% RSLogix 500 project Project6-HourMeter.RSS, saved by version 8.30.00.16 %
PROJECT "UNTITLED"    % processor: Bul.1763 MicroLogix 1100 Series B %

PROGRAM FILES
  LAD 2   8 rungs

DATA FILES
  O0 OUTPUT  4 elements
  I1 INPUT  6 elements
  S2 STATUS  66 elements
  B3 BINARY  1 elements
  T4 TIMER  1 elements
  C5 COUNTER  4 elements
  R6 CONTROL  1 elements
  N7 INTEGER  4 elements
  F8 FLOAT  1 elements

LADDER 2
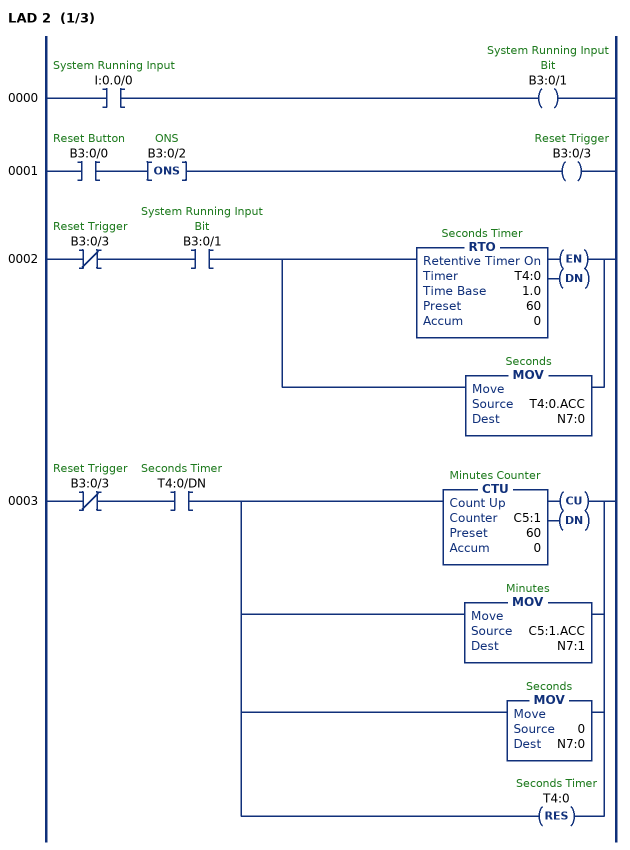
% Rung: 0 %
SOR XIC I:0.0/0 OTE B3:0/1 EOR
%   I:0.0/0  "System Running Input" %
%   B3:0/1  "System Running Input Bit" %
% Rung: 1 %  % edit flag set %
SOR XIC B3:0/0 ONS B3:0/2 OTE B3:0/3 EOR
%   B3:0/0  "Reset Button" %
%   B3:0/2  "ONS" %
%   B3:0/3  "Reset Trigger" %
% Rung: 2 %
SOR XIO B3:0/3 XIC B3:0/1 BST RTO T4:0 1.0 60 0 NXB MOV T4:0.ACC N7:0 BND EOR
%   B3:0/3  "Reset Trigger" %
%   B3:0/1  "System Running Input Bit" %
%   T4:0  "Seconds Timer" %
%   N7:0  "Seconds" %
% Rung: 3 %
SOR XIO B3:0/3 XIC T4:0/DN BST CTU C5:1 60 0 NXB MOV C5:1.ACC N7:1 NXB MOV 0 N7:0 NXB RES T4:0 BND EOR
%   B3:0/3  "Reset Trigger" %
%   T4:0  "Seconds Timer" %
%   C5:1  "Minutes Counter" %
%   N7:1  "Minutes" %
%   N7:0  "Seconds" %

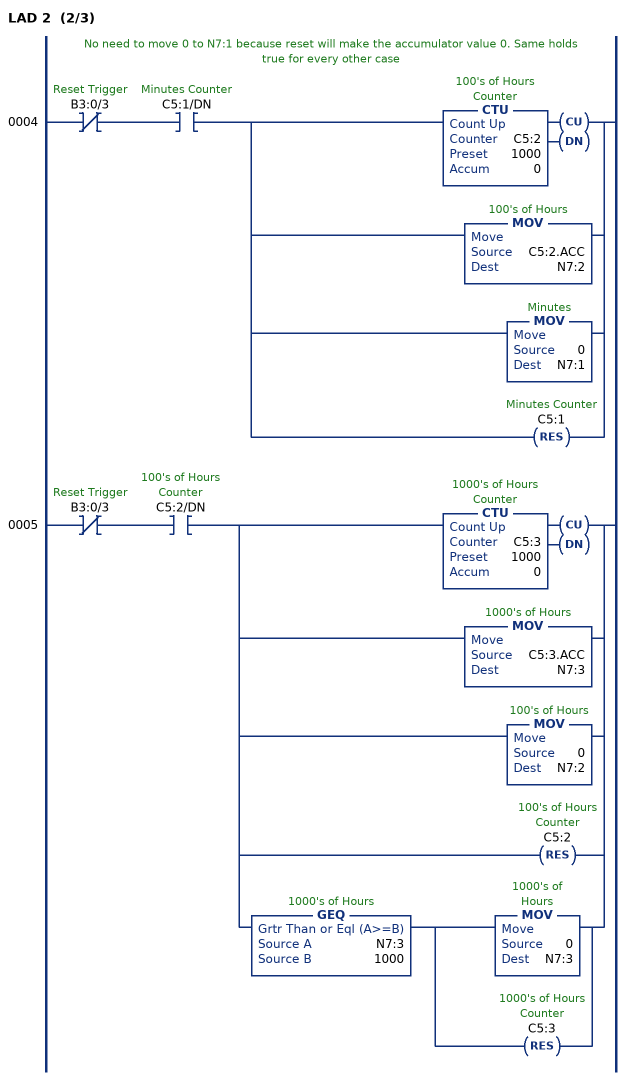
% Rung: 4 %
% No need to move 0 to N7:1 because reset will make the accumulator value 0. Same holds true for every other case %
SOR XIO B3:0/3 XIC C5:1/DN BST CTU C5:2 1000 0 NXB MOV C5:2.ACC N7:2 NXB MOV 0 N7:1 NXB RES C5:1 BND EOR
%   B3:0/3  "Reset Trigger" %
%   C5:1  "Minutes Counter" %
%   C5:2  "100's of Hours Counter" %
%   N7:2  "100's of Hours" %
%   N7:1  "Minutes" %
% Rung: 5 %  % edit flag set %
SOR XIO B3:0/3 XIC C5:2/DN BST CTU C5:3 1000 0 NXB MOV C5:3.ACC N7:3 NXB MOV 0 N7:2 NXB RES C5:2 NXB GEQ N7:3 1000 BST MOV 0 N7:3 NXB RES C5:3 BND BND EOR
%   B3:0/3  "Reset Trigger" %
%   C5:2  "100's of Hours Counter" %
%   C5:3  "1000's of Hours Counter" %
%   N7:3  "1000's of Hours" %
%   N7:2  "100's of Hours" %

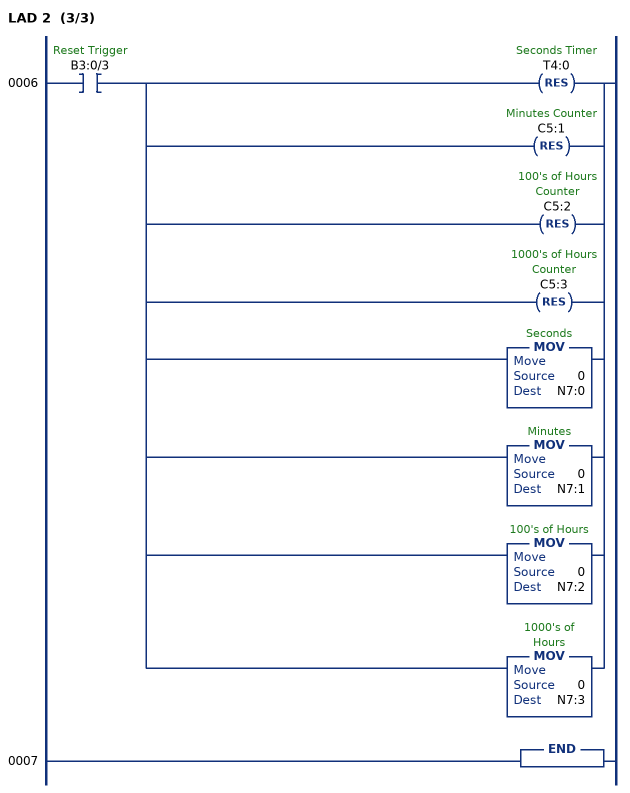
% Rung: 6 %
SOR XIC B3:0/3 BST RES T4:0 NXB RES C5:1 NXB RES C5:2 NXB RES C5:3 NXB MOV 0 N7:0 NXB MOV 0 N7:1 NXB MOV 0 N7:2 NXB MOV 0 N7:3 BND EOR
%   B3:0/3  "Reset Trigger" %
%   T4:0  "Seconds Timer" %
%   C5:1  "Minutes Counter" %
%   C5:2  "100's of Hours Counter" %
%   C5:3  "1000's of Hours Counter" %
%   N7:0  "Seconds" %
%   N7:1  "Minutes" %
%   N7:2  "100's of Hours" %
%   N7:3  "1000's of Hours" %
% Rung: 7 %
SOR END EOR

OTHER DOCUMENTED ADDRESSES
  C5:0  "Seconds Counter"

DATA TABLE (non-zero values as saved)
DATA B3
% B3:0 % 0X0005
DATA T4
% .PRE .ACC %
% T4:0 % 60 0
DATA C5
% .PRE .ACC %
% C5:1 % 60 0
% C5:2 % 1000 0
% C5:3 % 10000 0
